FUNCTION_BLOCK FB_ServerOpcUa
VAR_INPUT
END_VAR
VAR_OUTPUT
END_VAR
VAR
END_VAR

END_FUNCTION_BLOCK

(* stored: Version 1.1.0.1, ProductVersion 3.1.4024.11
   POU FB_ServerOpcUa: Id {e7b0a92e-6673-4460-843f-494f972b71f9}, SpecialFunc None *)
